(*
SPDX-FileCopyrightText: Â© 2026 Oleksandr Tiutyk <trofimich@gmail.com>
SPDX-License-Identifier: MIT
License: https://opensource.org/license/mit
*)

(*!
<summary>Defines simulation mode override behavior for child components.</summary>
<description>
Allows individual child components to follow the parent's simulation state or explicitly force simulation ON or OFF.
</description>
*)

{attribute 'qualified_only'}
{attribute 'strict'}
{attribute 'to_string'}
TYPE SIMULATION_MODE_OVERRIDE :
(
	(*! <summary>Inherit simulation mode from parent component.</summary> *)
	INHERITED := 0,
	(*! <summary>Force simulation mode ON regardless of parent setting.</summary> *)
	ON,
	(*! <summary>Force simulation mode OFF regardless of parent setting.</summary> *)
	OFF
);
END_TYPE

(* stored: Version 1.1.0.1
   DUT SIMULATION_MODE_OVERRIDE: Id {b8b8c23e-8b75-4049-b4d6-b0767b0f81a1} *)
